// TIA Portal V17 export
// export: Created 2026-07-18T06:00:00.0000000Z, ExportSetting WithDefaults
DATA_BLOCK "MotorFbInstance"   // DB2
{ S7_Optimized_Access := 'TRUE' }
VERSION : 0.1
// stored: AutoNumber true, InstanceOfName MotorFb, IsIECCheckEnabled false
"MotorFb"
   // VAR
   //    Running : Bool;
   //    Setpoint : Real;
   // END_VAR
BEGIN
END_DATA_BLOCK
